// TIA Portal V20 export
// export: Created 2025-12-01T15:00:13.3023197Z, ExportSetting None, DisplayName Totally Integrated Automation Portal, DisplayVersion V20 Update 3, DisplayName TIA Portal Openness, DisplayVersion V20 Update 3, DisplayName TIA Portal Version Control Interface, DisplayVersion V20 Update 3, DisplayName STEP 7 Professional, DisplayVersion V20 Update 3, DisplayName STEP 7 Safety, DisplayVersion V20 Update 2, DisplayName WinCC Basic/Comfort/Advanced, DisplayVersion V20 Update 3, DisplayName WinCC Professional, DisplayVersion V20 Update 3, DisplayName WinCC Unified, DisplayVersion V20 Update 3
DATA_BLOCK "DB856_TipoMesaPantalla"   // DB856
{ S7_Optimized_Access := 'FALSE' }
AUTHOR : PANTALLA
NAME : 20130301
VERSION : 3.0
// stored: AutoNumber false
   VAR RETAIN
      TipoMesa : Array[0.."CTE_MaxMesas"] of Struct
         Tipo { S7_SetPoint := 'True'} : "TipoMesaPantalla";   // Tipo de Mesa para configurar la pantalla
      END_STRUCT;
   END_VAR
BEGIN
END_DATA_BLOCK
